Yaskawa INFORM job: X2_104(180,0).JBI

/JOB
//NAME X2_104(180,0)
//POS
///NPOS 389,389,389,11,0,0
///TOOL 0
///POSTYPE PULSE
///PULSE
C00000=-2887,-122912,-116763,204,79921,-300
C00001=105948,-60265,-68612,15471,82266,-26774
C00002=105944,-60303,-65683,15533,80508,-26998
C00003=105943,-60263,-64482,15562,79814,-27086
C00004=105942,-60151,-62762,15605,78849,-27210
C00005=105943,-60263,-64482,15562,79814,-27086
C00006=105943,-60248,-64197,15569,79653,-27107
C00007=105943,-60248,-64195,15569,79652,-27108
C00008=105943,-60248,-64197,15569,79653,-27107
C00009=105943,-60248,-64197,15569,79653,-27107
C00010=105942,-60174,-63048,15598,79008,-27190
C00011=105941,-60184,-63045,15598,79001,-27191
C00012=105942,-60174,-63048,15598,79008,-27190
C00013=105943,-60249,-64198,15569,79653,-27107
C00014=105943,-60263,-64482,15562,79814,-27086
C00015=105944,-60303,-65683,15533,80508,-26998
C00016=105948,-60265,-68612,15471,82266,-26774
C00017=109877,-64973,-75760,9490,93075,-21209
C00018=144619,-68543,-73003,-20989,87470,27722
C00019=149622,-57030,-60721,-30956,83108,29784
C00020=149622,-56790,-58217,-31031,81883,30116
C00021=149622,-56662,-57196,-31066,81398,30250
C00022=149623,-56407,-55393,-31134,80554,30482
C00023=149622,-56662,-57196,-31066,81398,30250
C00024=150587,-55933,-56592,-31222,81757,30533
C00025=149619,-56625,-56981,-31073,81300,30276
C00026=149621,-56633,-56977,-31074,81295,30278
C00027=149622,-56635,-56981,-31074,81296,30278
C00028=149617,-56657,-57316,-31061,81462,30231
C00029=149617,-56657,-57313,-31061,81461,30231
C00030=149617,-56657,-57316,-31061,81462,30231
C00031=149622,-56635,-56981,-31074,81296,30278
C00032=149622,-56662,-57196,-31066,81398,30250
C00033=149622,-56790,-58217,-31031,81883,30116
C00034=149622,-57030,-60721,-30956,83108,29784
C00035=144619,-68543,-73003,-20989,87470,27722
C00036=114895,-83747,-80366,6772,73338,-8124
C00037=115460,-69444,-73725,6516,76534,-7754
C00038=115459,-69304,-70716,6562,74765,-7849
C00039=115458,-69195,-69485,6584,74068,-7887
C00040=115458,-68988,-67720,6614,73094,-7940
C00041=115458,-69195,-69485,6584,74068,-7887
C00042=115458,-69074,-68335,6603,73428,-7921
C00043=115457,-69075,-68332,6603,73425,-7921
C00044=115458,-69074,-68335,6603,73428,-7921
C00045=115458,-69210,-69581,6582,74119,-7884
C00046=115459,-69422,-72626,6532,75874,-7789
C00047=114895,-83747,-80366,6772,73338,-8124
C00048=122568,-82719,-80422,-802,72905,572
C00049=122404,-70386,-74693,-742,75716,497
C00050=122404,-70253,-71692,-748,73937,507
C00051=122404,-70146,-70463,-750,73236,512
C00052=122404,-69945,-68703,-754,72256,518
C00053=122404,-70146,-70463,-750,73236,512
C00054=122403,-69999,-69129,-754,72490,516
C00055=122403,-69999,-69126,-754,72489,516
C00056=122403,-69999,-69129,-754,72490,516
C00057=122426,-71764,-70432,-761,72385,525
C00058=125366,-69810,-69017,-1661,72563,1552
C00059=139732,-60008,-63655,-19169,79951,16701
C00060=138795,-60432,-63881,-18965,79660,16411
C00061=141372,-63440,-66071,-19537,80074,17269
C00062=131414,-76802,-75559,-9437,74661,8207
C00063=122633,-87524,-80325,-832,70378,611
C00064=122404,-70253,-71692,-748,73937,507
C00065=122404,-70386,-74693,-742,75716,497
C00066=122568,-82719,-80422,-802,72905,572
C00067=120793,-80683,-79694,968,73556,-1433
C00068=120782,-70088,-74721,961,75940,-1419
C00069=120781,-69974,-71726,968,74156,-1433
C00070=120781,-69875,-70501,972,73453,-1438
C00071=120781,-69685,-68746,976,72471,-1446
C00072=120781,-69875,-70501,972,73453,-1438
C00073=120781,-69719,-69028,976,72627,-1445
C00074=120781,-69719,-69024,976,72624,-1446
C00075=120781,-69719,-69028,976,72627,-1445
C00076=120781,-69868,-70316,972,73342,-1439
C00077=121987,-69893,-70664,604,73531,-1018
C00078=120781,-69902,-70677,972,73547,-1437
C00079=120781,-69912,-70673,972,73540,-1437
C00080=120781,-69738,-69020,976,72612,-1445
C00081=120781,-69875,-70501,972,73453,-1438
C00082=120781,-69974,-71726,968,74156,-1433
C00083=120782,-70088,-74721,961,75940,-1419
C00084=109767,-94679,-77625,-554,64647,-3819
C00085=110036,-87261,-71666,-642,64793,-3719
C00086=110147,-84282,-69219,-679,64819,-3677
C00087=106931,-83315,-68824,372,65076,-4870
C00088=120553,-76872,-65939,-13890,70696,12122
C00089=123092,-73013,-64238,-16293,73991,15774
C00090=123502,-72820,-64152,-16860,74575,16660
C00091=130441,-60579,-57109,-23338,83277,32357
C00092=128852,-72596,-62262,-22941,75556,33354
C00093=130317,-73839,-64199,-23146,76478,33722
C00094=133782,-77123,-68532,-23639,78364,34645
C00095=137012,-102538,-78858,-24747,73168,36952
C00096=156868,-82779,-69870,-33497,82961,10620
C00097=152555,-67883,-62928,-32980,84120,8538
C00098=153259,-66149,-60215,-33082,83738,8932
C00099=149912,-60899,-55666,-32717,82430,7997
C00100=128127,-81205,-68774,-8858,64404,-8706
C00101=128406,-81696,-69061,-3569,63264,-13044
C00102=126372,-87795,-73203,-2830,62599,-13791
C00103=116888,-93582,-79828,8557,66782,-12634
C00104=92924,-89512,-73118,32406,78401,-8719
C00105=72721,-73373,-69592,26022,86972,-15267
C00106=80895,-52896,-59408,25141,88320,-11942
C00107=83138,-49043,-54251,24862,86564,-11488
C00108=85205,-49270,-53237,24600,85277,-10995
C00109=85821,-49873,-53436,24520,84922,-10841
C00110=95949,-62919,-60694,23037,79963,-8102
C00111=102091,-71911,-65157,19247,73237,-2273
C00112=116516,-77081,-67507,13716,67864,4585
C00113=112851,-78661,-66635,20192,66100,7115
C00114=125798,-85436,-69237,6250,57352,21558
C00115=146063,-75361,-64399,-19160,63709,45094
C00116=156433,-45058,-47672,-31921,84708,61878
C00117=158375,-58932,-51564,-37026,71970,66054
C00118=159846,-59274,-53202,-37172,73275,66233
C00119=163234,-59592,-56142,-37574,76069,66714
C00120=168472,-71553,-64044,-35465,82568,67157
C00121=118088,-113838,-85475,7366,65299,-32947
C00122=118732,-79947,-72555,6808,74639,-32160
C00123=121034,-75641,-67247,6295,73405,-31417
C00124=122088,-73495,-65040,6051,73071,-31063
C00125=121942,-71052,-63825,6072,73586,-31087
C00126=123099,-75779,-64750,4483,66211,-39428
C00127=121321,-81189,-67590,5597,62405,-44748
C00128=118846,-85423,-72852,6459,63648,-45617
C00129=118212,-118410,-84702,7387,54112,-46472
C00130=-871,-167382,-128748,-2443,88873,-10065
C00131=-871,-167382,-128748,-2443,88873,-10065
C00132=57381,82979,10637,-12644,90379,68932
C00133=127807,-61304,-68748,-13816,80064,24242
C00134=125765,-61582,-65964,-13370,77922,23771
C00135=124946,-61609,-64807,-13191,77080,23576
C00136=124950,-61468,-63072,-13241,76110,23683
C00137=124946,-61609,-64807,-13191,77080,23576
C00138=124976,-61587,-64521,-13207,76925,23603
C00139=124980,-61587,-64530,-13208,76931,23604
C00140=124976,-61587,-64521,-13207,76925,23603
C00141=124935,-61591,-64522,-13196,76916,23590
C00142=124937,-61496,-63363,-13229,76268,23661
C00143=123116,-61640,-63435,-12754,75950,23053
C00144=124937,-61496,-63363,-13229,76268,23661
C00145=124935,-61591,-64522,-13196,76916,23590
C00146=124946,-61609,-64807,-13191,77080,23576
C00147=125765,-61582,-65964,-13370,77922,23771
C00148=127807,-61304,-68748,-13816,80064,24242
C00149=123100,-60794,-73195,-8642,92314,18302
C00150=97511,-77513,-76888,20898,84915,-28039
C00151=93556,-58201,-60930,30710,81826,-29583
C00152=93550,-57951,-58428,30804,80607,-29915
C00153=93548,-57820,-57410,30845,80124,-30048
C00154=93546,-57539,-55590,30923,79282,-30278
C00155=93548,-57820,-57410,30845,80124,-30048
C00156=93547,-57790,-57188,30855,80020,-30076
C00157=93545,-57800,-57196,30855,80021,-30077
C00158=93547,-57790,-57188,30855,80020,-30076
C00159=93548,-57786,-57169,30855,80012,-30078
C00160=93543,-57856,-57518,30843,80168,-30037
C00161=93543,-57857,-57528,30842,80172,-30036
C00162=93543,-57856,-57518,30843,80168,-30037
C00163=93548,-57786,-57169,30855,80012,-30078
C00164=93548,-57820,-57410,30845,80124,-30048
C00165=93550,-57951,-58428,30804,80607,-29915
C00166=93556,-58201,-60930,30710,81826,-29583
C00167=97511,-77513,-76888,20898,84915,-28039
C00168=129623,-93566,-83802,-7941,70327,9276
C00169=128126,-69066,-72890,-7284,76011,8392
C00170=128127,-68885,-69881,-7338,74266,8496
C00171=128227,-70585,-69547,-7404,73204,8596
C00172=128227,-70369,-67888,-7439,72303,8652
C00173=128262,-71214,-69852,-7419,73073,8616
C00174=128200,-69934,-68140,-7416,72675,8619
C00175=128127,-68612,-67496,-7384,72949,8576
C00176=128127,-68613,-67489,-7384,72944,8577
C00177=128127,-68764,-68733,-7360,73627,8535
C00178=128126,-69014,-71778,-7303,75358,8431
C00179=129623,-93566,-83802,-7941,70327,9276
C00180=121374,-102449,-87359,-63,66651,180
C00181=121222,-71970,-74483,-14,74388,124
C00182=121222,-71735,-71450,-14,72642,124
C00183=121228,-73354,-70977,-16,71518,126
C00184=121228,-73077,-69260,-16,70604,126
C00185=121230,-73832,-71281,-16,71462,127
C00186=121229,-73317,-69774,-16,70798,128
C00187=121222,-71403,-68866,-14,71222,125
C00188=121222,-71402,-68857,-14,71217,125
C00189=121222,-71370,-68825,-14,71214,125
C00190=121222,-71504,-69842,-14,71771,124
C00191=121222,-71516,-69850,-14,71770,124
C00192=121222,-71504,-69842,-14,71771,124
C00193=121222,-71598,-70490,-14,72121,125
C00194=121222,-71590,-70211,-14,71954,124
C00195=121222,-71735,-71450,-14,72642,124
C00196=121222,-71970,-74483,-14,74388,124
C00197=121374,-102449,-87359,-63,66651,180
C00198=123521,-105913,-88673,-2044,65797,2436
C00199=122862,-71970,-74551,-1739,74528,2064
C00200=122862,-71740,-71520,-1753,72781,2089
C00201=122863,-71596,-70280,-1759,72093,2099
C00202=122863,-71343,-68495,-1768,71124,2113
C00203=122863,-71596,-70280,-1759,72093,2099
C00204=122863,-71387,-68782,-1767,71278,2111
C00205=122863,-71388,-68789,-1767,71282,2111
C00206=122863,-71387,-68782,-1767,71278,2111
C00207=122862,-71560,-70082,-1760,71989,2100
C00208=122862,-71596,-70456,-1758,72201,2098
C00209=122862,-71608,-70465,-1758,72201,2098
C00210=122862,-71596,-70456,-1758,72201,2098
C00211=122862,-71364,-68762,-1767,71278,2111
C00212=122863,-71596,-70280,-1759,72093,2099
C00213=122862,-71740,-71520,-1753,72781,2089
C00214=122862,-71970,-74551,-1739,74528,2064
C00215=133853,-94891,-77624,-322,64195,4510
C00216=133469,-87446,-71679,-193,64361,4366
C00217=133332,-84612,-69279,-149,64338,4316
C00218=136520,-83360,-68727,-1205,64680,5498
C00219=122681,-77523,-66172,13350,69902,-11676
C00220=120168,-73612,-64489,15807,73184,-15339
C00221=112575,-61593,-57739,23052,82443,-32062
C00222=113938,-70945,-61811,22691,76593,-32754
C00223=112608,-75313,-64851,22854,75462,-33489
C00224=109132,-78771,-69243,23377,77292,-34432
C00225=105658,-108562,-80888,24788,70838,-37103
C00226=81640,-97499,-76087,33945,80765,-12609
C00227=90241,-69606,-64048,32870,83199,-8395
C00228=92951,-64963,-58962,32610,81520,-7798
C00229=93939,-63321,-57029,32518,80848,-7597
C00230=125857,-77866,-68310,-6550,68061,3456
C00231=123054,-78148,-68482,-5670,67810,2448
C00232=143027,-65706,-58192,-31754,78539,6334
C00233=144021,-67708,-60230,-31872,79107,6572
C00234=146628,-72736,-65452,-32167,80634,7181
C00235=152532,-96040,-75422,-33296,77968,10353
C00236=170079,-74119,-69784,-26506,86877,15660
C00237=161776,-50684,-58065,-25622,88646,12176
C00238=159526,-46913,-52939,-25338,86859,11731
C00239=158170,-45955,-51438,-25163,86055,11404
C00240=157195,-47475,-52284,-25036,85525,11154
C00241=146543,-61011,-59669,-23472,80213,8306
C00242=141963,-69014,-63758,-20053,74078,2973
C00243=126831,-75909,-66940,-14438,68034,-4018
C00244=130165,-77618,-66175,-20834,66320,-6667
C00245=117599,-84808,-69026,-7184,57298,-20899
C00246=97281,-75815,-64687,18602,62898,-44607
C00247=86271,-46211,-48696,31805,84024,-61698
C00248=85005,-58470,-51696,36499,71620,-65497
C00249=82871,-59517,-53345,37068,72494,-66094
C00250=79472,-59950,-56347,37489,75274,-66588
C00251=72756,-72734,-64617,35623,82237,-67485
C00252=121023,-109349,-83964,-6868,66067,31929
C00253=120934,-78788,-71982,-6517,74337,31434
C00254=118696,-74387,-66630,-5999,73137,30708
C00255=117510,-72864,-64443,-5724,72490,30318
C00256=117903,-69871,-63138,-5800,73250,30422
C00257=117006,-77674,-64461,-4475,61816,43275
C00258=118051,-79909,-67055,-4889,62200,43848
C00259=120454,-84253,-72369,-5752,63392,44701
C00260=120394,-115928,-83972,-6293,54299,45179
C00261=-2019,-116841,-84248,8,53945,-8
C00262=-2019,-116841,-84248,8,53945,-8
C00263=73594,47215,-15331,-17682,89066,63909
C00264=142113,-97158,-104646,-26332,80699,28696
C00265=126900,-111905,-82922,-22333,65135,26241
C00266=123037,-105645,-78013,-21421,64295,24879
C00267=121585,-103154,-76020,-21064,63971,24366
C00268=121574,-101968,-73872,-21184,63301,24491
C00269=121585,-103154,-76020,-21064,63971,24366
C00270=121605,-102291,-74338,-21170,63423,24480
C00271=121584,-98936,-73211,-20991,64381,24287
C00272=121605,-102291,-74338,-21170,63423,24480
C00273=121452,-100284,-74443,-20948,64409,24229
C00274=118901,-100253,-74439,-20311,63782,23339
C00275=121452,-100284,-74443,-20948,64409,24229
C00276=122866,-102731,-76445,-21292,64747,24723
C00277=126621,-108872,-81370,-22171,65621,26033
C00278=121330,-115088,-85498,-358,58030,151
C00279=121291,-106557,-79734,-341,58867,134
C00280=121277,-103287,-77415,-334,59121,127
C00281=121267,-102136,-75285,-334,58400,125
C00282=121277,-103287,-77415,-334,59121,127
C00283=121242,-102632,-75811,-324,58469,116
C00284=121234,-99223,-74662,-318,59514,110
C00285=121242,-102632,-75811,-324,58469,116
C00286=121256,-105876,-78126,-330,58227,122
C00287=121292,-114324,-83876,-346,57425,139
C00288=121322,-115349,-85447,-355,57865,149
C00289=121283,-106809,-79688,-338,58709,131
C00290=121269,-103536,-77371,-332,58965,124
C00291=121259,-102375,-75237,-331,58248,123
C00292=121269,-103536,-77371,-332,58965,124
C00293=121253,-102639,-75604,-329,58338,121
C00294=121245,-99239,-74459,-322,59381,114
C00295=121253,-102639,-75604,-329,58338,121
C00296=121268,-105882,-77919,-334,58096,127
C00297=121305,-114323,-83666,-351,57296,144
C00298=121318,-115477,-85353,-354,57741,148
C00299=121280,-106935,-79598,-338,58589,130
C00300=121266,-103662,-77282,-331,58845,124
C00301=121256,-102495,-75146,-331,58130,122
C00302=121266,-103662,-77282,-331,58845,124
C00303=121259,-102859,-75577,-331,58209,124
C00304=121251,-99462,-74437,-325,59253,117
C00305=121259,-102859,-75577,-331,58209,124
C00306=121274,-106105,-77890,-337,57965,130
C00307=121311,-114553,-83633,-354,57157,147
C00308=121337,-115746,-85310,-361,57577,156
C00309=121297,-107196,-79560,-344,58432,137
C00310=121283,-103917,-77246,-338,58692,131
C00311=121272,-102742,-75106,-337,57980,130
C00312=121283,-103917,-77246,-338,58692,131
C00313=121246,-102874,-75436,-326,58114,118
C00314=121237,-99483,-74299,-320,59157,112
C00315=121246,-102874,-75436,-326,58114,118
C00316=121259,-106119,-77748,-333,57870,124
C00317=121296,-114563,-83488,-348,57063,142
C00318=115780,-112688,-82708,21819,64400,-26075
C00319=119618,-106339,-77769,20890,63616,-24706
C00320=121058,-103816,-75763,20529,63312,-24192
C00321=121048,-102603,-73605,20653,62653,-24321
C00322=121058,-103816,-75763,20529,63312,-24192
C00323=121040,-102752,-73855,20641,62728,-24310
C00324=121038,-99421,-72747,20466,63695,-24129
C00325=121040,-102752,-73855,20641,62728,-24310
C00326=118303,-96965,-72660,22305,67146,-26975
C00327=118267,-92509,-70963,23513,70285,-29122
C00328=120824,-100634,-73993,20495,63883,-24177
C00329=119419,-103098,-76004,20840,64209,-24672
C00330=115684,-109288,-80956,21727,65048,-25985
C00331=96888,-111476,-87068,9061,72855,-9977
C00332=98574,-104492,-81262,8787,72684,-9391
C00333=93909,-110684,-79514,13666,64171,-14539
C00334=141627,-111255,-79468,4808,59529,5267
C00335=116884,-104836,-72389,32528,66157,393
C00336=116227,-100796,-73717,31025,72452,2000
C00337=113714,-107379,-79275,31259,73409,1253
C00338=145516,-110399,-87018,-9521,73555,10095
C00339=143792,-103507,-81225,-9247,73331,9501
C00340=147991,-116725,-79770,-15189,57547,12945
C00341=92805,-108670,-79244,2926,60987,-8726
C00342=125500,-104465,-72202,-33294,65779,-22
C00343=126155,-100219,-73727,-31459,72916,-1934
C00344=128707,-106743,-79266,-31688,73916,-1183
C00345=149163,-107491,-85659,-10054,74646,11300
C00346=147320,-100877,-79905,-9779,74280,10678
C00347=149405,-108030,-78804,-12916,65248,12387
C00348=93726,-109350,-79423,2686,60646,-8385
C00349=95575,-101419,-80230,-67,70891,-7504
C00350=94880,-108692,-86195,76,70825,-7751
C00351=93512,-107502,-86110,9531,74678,-11036
C00352=95285,-100847,-80339,9259,74342,-10434
C00353=91829,-111238,-79018,14022,61540,-13112
C00354=149361,-109410,-78888,-3377,59825,8868
C00355=152861,-110027,-78581,-5464,58492,10359
C00356=146783,-100727,-80168,-430,71345,7655
C00357=147530,-107934,-86130,-582,71316,7920
C00358=147530,-109971,-90893,-577,73200,7911
C00359=147530,-109971,-90893,-577,73200,7911
C00360=129338,-115306,-83649,32043,62659,-1447
C00361=109985,-114895,-67593,57991,58611,-29778
C00362=123189,-110825,-64198,56881,47665,-25598
C00363=123974,-108354,-57257,59191,45569,-26987
C00364=133588,-111477,-65669,41012,44431,-18914
C00365=131723,-121473,-78996,33426,49678,-16861
C00366=131723,-127083,-87093,32500,51454,-16199
C00367=112124,-99575,-74661,44559,72636,-57535
C00368=144481,-87729,-76760,13160,69523,-45180
C00369=143253,-81512,-73231,13426,70725,-45494
C00370=141746,-72876,-67816,13764,72050,-45890
C00371=140405,-91076,-80988,14230,71070,-46496
C00372=147724,-115880,-117962,-4434,76384,7704
C00373=102175,-95850,-84882,-8811,63963,-9409
C00374=106773,-75463,-61467,-29853,53349,18924
C00375=99131,-70118,-56440,-22082,48330,13186
C00376=98320,-68106,-55033,-21545,48270,12812
C00377=98199,-68741,-54193,-21751,47452,12950
C00378=97569,-68978,-50300,-22280,44856,13272
C00379=93899,-57457,-51708,-11926,60791,9289
C00380=97609,-69104,-63179,-12714,63588,10475
C00381=100380,-33173,-52064,-13535,85135,38620
C00382=91620,-26640,-46583,-3556,85730,36721
C00383=94429,-23251,-43461,-7027,86025,37207
C00384=96713,-17180,-36687,-8408,83804,38028
C00385=103963,-23375,-42130,-14397,84680,39883
C00386=111815,-38667,-59152,-16138,88632,42049
C00387=147724,-115880,-117962,-4434,76384,7704
C00388=-2019,-116841,-84248,8,53945,-8
BC00000=780,523905,878730
BC00001=24680,466753,17
BC00002=21091,462611,17
BC00003=19655,460955,17
BC00004=19671,460959,17
BC00005=19655,460955,17
BC00006=19705,460415,17
BC00007=19697,457343,17
BC00008=19705,460415,17
BC00009=19637,460956,17
BC00010=19648,460935,17
BC00011=16462,460942,17
BC00012=19648,460935,17
BC00013=19637,460956,17
BC00014=19655,460955,17
BC00015=21091,462611,17
BC00016=24680,466753,17
BC00017=23714,465651,17
BC00018=75244,465786,17
BC00019=74371,466642,17
BC00020=78995,462188,17
BC00021=80845,460407,17
BC00022=80861,460411,17
BC00023=80845,460407,17
BC00024=81362,460408,17
BC00025=84547,460400,17
BC00026=81362,460408,17
BC00027=80862,466105,17
BC00028=88196,466087,17
BC00029=88188,463015,17
BC00030=88196,466087,17
BC00031=80862,466105,17
BC00032=80845,460407,17
BC00033=78995,462188,17
BC00034=74371,466642,17
BC00035=75244,465786,17
BC00036=130207,468776,17
BC00037=130207,468776,17
BC00038=128970,463491,17
BC00039=128475,461377,17
BC00040=128491,461381,17
BC00041=128475,461377,17
BC00042=126183,462269,17
BC00043=125467,459275,17
BC00044=126183,462269,17
BC00045=126677,464383,17
BC00046=127915,469668,17
BC00047=130207,468776,17
BC00048=334579,467175,17
BC00049=334579,467175,17
BC00050=334594,461751,17
BC00051=334599,459581,17
BC00052=334616,459585,17
BC00053=334599,459581,17
BC00054=334621,459509,17
BC00055=334613,456436,17
BC00056=334621,459509,17
BC00057=326309,462655,17
BC00058=326309,462655,17
BC00059=323407,460034,17
BC00060=323407,460034,17
BC00061=323407,460034,17
BC00062=325115,461032,17
BC00063=334599,459581,17
BC00064=334594,461751,17
BC00065=334579,467175,17
BC00066=334579,467175,17
BC00067=391469,467628,17
BC00068=391469,467628,17
BC00069=391192,462215,17
BC00070=391081,460050,17
BC00071=391097,460054,17
BC00072=391081,460050,17
BC00073=391084,460088,17
BC00074=390911,457021,17
BC00075=391084,460088,17
BC00076=387971,461309,17
BC00077=384628,457146,17
BC00078=387809,456979,17
BC00079=384628,457146,17
BC00080=384826,460381,17
BC00081=391081,460050,17
BC00082=391192,462215,17
BC00083=391469,467628,17
BC00084=363156,441715,38776
BC00085=363156,441715,38776
BC00086=363156,441715,38776
BC00087=363156,441715,38776
BC00088=363156,441715,38776
BC00089=363156,441715,38776
BC00090=363156,441715,38776
BC00091=363156,441715,38776
BC00092=363156,441715,38776
BC00093=363156,441715,38776
BC00094=363156,441715,38776
BC00095=363156,441715,38776
BC00096=338596,448628,25253
BC00097=338596,448628,25253
BC00098=338596,448628,25253
BC00099=338597,448627,25252
BC00100=338597,448627,25252
BC00101=338597,448627,25252
BC00102=338597,448627,25252
BC00103=338597,448627,25252
BC00104=338596,448628,25253
BC00105=96993,454866,20869
BC00106=98278,457002,17644
BC00107=98278,457002,17644
BC00108=98278,457002,17644
BC00109=98278,457002,17644
BC00110=98278,457002,17644
BC00111=98278,457002,17644
BC00112=98278,457002,17644
BC00113=98278,457002,17644
BC00114=98278,457002,17644
BC00115=98278,457002,17644
BC00116=98278,457002,17644
BC00117=98278,457002,17644
BC00118=98278,457002,17644
BC00119=98278,457002,17644
BC00120=96993,454866,20869
BC00121=35692,446449,44492
BC00122=35692,446449,44492
BC00123=35692,446449,44492
BC00124=35692,446449,44492
BC00125=35692,446449,44492
BC00126=35692,446449,44492
BC00127=35692,446449,44492
BC00128=35692,446449,44492
BC00129=35692,446449,44492
BC00130=226112,522070,21179
BC00131=226112,522070,21179
BC00132=201604,630124,773856
BC00133=397680,544373,17
BC00134=397680,461002,17
BC00135=397680,459324,17
BC00136=397680,459307,17
BC00137=397680,459324,17
BC00138=397680,458781,17
BC00139=397680,455709,17
BC00140=397680,458781,17
BC00141=397680,459321,17
BC00142=397680,459287,17
BC00143=397680,459279,17
BC00144=397680,459287,17
BC00145=397680,459321,17
BC00146=397680,459324,17
BC00147=397680,461002,17
BC00148=397680,465197,17
BC00149=397680,464098,17
BC00150=364002,464474,17
BC00151=364885,465316,17
BC00152=360253,460854,17
BC00153=358400,459070,17
BC00154=358395,459053,17
BC00155=358400,459070,17
BC00156=357885,459071,17
BC00157=354700,459079,17
BC00158=357885,459071,17
BC00159=358414,464766,17
BC00160=351078,464787,17
BC00161=351070,461715,17
BC00162=351078,464787,17
BC00163=358414,464766,17
BC00164=358400,459070,17
BC00165=360253,460854,17
BC00166=364885,465316,17
BC00167=364002,464474,17
BC00168=309055,467727,17
BC00169=309055,467727,17
BC00170=310284,462400,17
BC00171=310775,460269,17
BC00172=310770,460253,17
BC00173=310775,460269,17
BC00174=313079,461137,17
BC00175=313780,458140,17
BC00176=313079,461137,17
BC00177=312588,463268,17
BC00178=311359,468595,17
BC00179=309055,467727,17
BC00180=104675,467109,17
BC00181=104675,467109,17
BC00182=104651,461649,17
BC00183=104636,459449,17
BC00184=104636,459449,17
BC00185=104642,459465,17
BC00186=104628,459377,17
BC00187=104620,456305,17
BC00188=104628,459377,17
BC00189=112956,462483,17
BC00190=116212,459519,17
BC00191=113027,459526,17
BC00192=116212,459519,17
BC00193=112864,461621,17
BC00194=104642,459465,17
BC00195=104651,461649,17
BC00196=104675,467109,17
BC00197=104675,467109,17
BC00198=47788,467835,17
BC00199=47788,467835,17
BC00200=48056,462385,17
BC00201=48163,460205,17
BC00202=48157,460188,17
BC00203=48163,460205,17
BC00204=48169,460226,17
BC00205=48326,457158,17
BC00206=48169,460226,17
BC00207=51281,461447,17
BC00208=54599,457272,17
BC00209=51418,457121,17
BC00210=54599,457272,17
BC00211=54429,460489,17
BC00212=48163,460205,17
BC00213=48056,462385,17
BC00214=47788,467835,17
BC00215=75364,442731,32628
BC00216=75364,442731,32628
BC00217=75364,442731,32628
BC00218=75364,442731,32628
BC00219=75364,442731,32628
BC00220=75364,442731,32628
BC00221=75364,442731,32628
BC00222=75364,442731,32628
BC00223=75364,442731,32628
BC00224=75364,442731,32628
BC00225=75364,442731,32628
BC00226=99841,449109,19074
BC00227=99841,449109,19074
BC00228=99841,449109,19074
BC00229=99841,449109,19074
BC00230=99841,449109,19074
BC00231=99841,449109,19074
BC00232=99841,449109,19074
BC00233=99841,449109,19074
BC00234=99841,449109,19074
BC00235=99841,449109,19074
BC00236=339958,454510,16791
BC00237=340496,456637,13010
BC00238=340496,456637,13010
BC00239=340496,456637,13010
BC00240=340496,456637,13010
BC00241=340496,456637,13010
BC00242=340496,456637,13010
BC00243=340496,456637,13010
BC00244=340496,456637,13010
BC00245=340496,456637,13010
BC00246=340496,456637,13010
BC00247=340496,456637,13010
BC00248=340496,456637,13010
BC00249=340496,456637,13010
BC00250=340496,456637,13010
BC00251=339958,454510,16791
BC00252=397680,444887,42686
BC00253=397680,444887,42686
BC00254=397680,444887,42686
BC00255=397680,444887,42686
BC00256=397680,444887,42686
BC00257=397680,444887,42686
BC00258=397680,444887,42686
BC00259=397680,444887,42686
BC00260=397680,444887,42686
BC00261=262396,523905,990511
BC00262=262396,523905,990511
BC00263=128960,592658,1075149
BC00264=336620,434807,1075139
BC00265=336620,389215,1075139
BC00266=336620,389215,1075139
BC00267=336620,389215,1075139
BC00268=336620,389215,1075139
BC00269=336620,389215,1075139
BC00270=336620,389215,1075139
BC00271=336620,389215,1075139
BC00272=336620,389215,1075139
BC00273=336620,389215,1075139
BC00274=336620,389215,1075139
BC00275=336620,389215,1075139
BC00276=336620,389215,1075139
BC00277=336620,389215,1075139
BC00278=314467,401738,1075139
BC00279=314467,401738,1075139
BC00280=314467,401738,1075139
BC00281=314467,401738,1075139
BC00282=314467,401738,1075139
BC00283=314467,401738,1075139
BC00284=314467,401738,1075139
BC00285=314467,401738,1075139
BC00286=314467,401738,1075139
BC00287=314467,401738,1075139
BC00288=250431,402103,1075139
BC00289=250431,402103,1075139
BC00290=250431,402103,1075139
BC00291=250431,402103,1075139
BC00292=250431,402103,1075139
BC00293=250431,402103,1075139
BC00294=250431,402103,1075139
BC00295=250431,402103,1075139
BC00296=250431,402103,1075139
BC00297=250431,402103,1075139
BC00298=181730,402292,1075139
BC00299=181730,402292,1075139
BC00300=181730,402292,1075139
BC00301=181730,402292,1075139
BC00302=181730,402292,1075139
BC00303=181730,402292,1075139
BC00304=181730,402292,1075139
BC00305=181730,402292,1075139
BC00306=181730,402292,1075139
BC00307=181730,402292,1075139
BC00308=120634,402626,1075139
BC00309=120634,402626,1075139
BC00310=120634,402626,1075139
BC00311=120634,402626,1075139
BC00312=120634,402626,1075139
BC00313=120634,402626,1075139
BC00314=120634,402626,1075139
BC00315=120634,402626,1075139
BC00316=120634,402626,1075139
BC00317=120634,402626,1075139
BC00318=98246,390680,1075139
BC00319=98246,390680,1075139
BC00320=98246,390680,1075139
BC00321=98246,390680,1075139
BC00322=98246,390680,1075139
BC00323=98246,390680,1075139
BC00324=98246,390680,1075139
BC00325=98246,390680,1075139
BC00326=98246,390680,1075139
BC00327=98246,390680,1075139
BC00328=98246,390680,1075139
BC00329=98246,390680,1075139
BC00330=98246,390680,1075139
BC00331=102602,381344,1075139
BC00332=102602,381344,1075139
BC00333=102602,381344,1075139
BC00334=102602,381344,1075139
BC00335=102602,381344,1075139
BC00336=102602,381344,1075139
BC00337=102602,381344,1075139
BC00338=332399,380541,1075139
BC00339=332399,380541,1075139
BC00340=332399,380541,1075139
BC00341=332399,380541,1075139
BC00342=332399,380541,1075139
BC00343=332399,380541,1075139
BC00344=332399,380541,1075139
BC00345=143465,382402,1075139
BC00346=143465,382402,1075139
BC00347=143465,382402,1075139
BC00348=143465,382402,1075139
BC00349=143465,382402,1075139
BC00350=143465,382402,1075139
BC00351=291477,381910,1075139
BC00352=291477,381910,1075139
BC00353=291477,381910,1075139
BC00354=291477,381910,1075139
BC00355=291477,381910,1075139
BC00356=291477,381910,1075139
BC00357=291477,381910,1075139
BC00358=291477,381910,1075139
BC00359=130464,381910,1075139
BC00360=130464,381910,1075139
BC00361=130464,381910,1075139
BC00362=130464,381910,1075139
BC00363=130464,381910,1075139
BC00364=130464,381910,1075139
BC00365=130464,381910,1075139
BC00366=130464,381910,1075139
BC00367=130464,381910,1075139
BC00368=130464,381910,1075139
BC00369=130464,381910,1075139
BC00370=130464,381910,1075139
BC00371=130464,381910,1075139
BC00372=291477,429847,1075139
BC00373=290233,429476,1075139
BC00374=290233,429476,1075139
BC00375=290233,429476,1075139
BC00376=290233,429476,1075139
BC00377=290233,429476,1075139
BC00378=290233,429476,1075139
BC00379=290233,429476,1075139
BC00380=290233,429476,1075139
BC00381=290234,429477,1075136
BC00382=290234,429477,1075136
BC00383=290234,429477,1075136
BC00384=290234,429477,1075136
BC00385=290234,429477,1075136
BC00386=290234,429477,1075136
BC00387=291477,429847,1075139
BC00388=262396,523905,990511
EC00000=-1596313,-183832
EC00001=-1596313,-183832
EC00002=-1596313,-183832
EC00003=-1596313,-183832
EC00004=-1596313,-183832
EC00005=-1596313,-183832
EC00006=-1596313,-183832
EC00007=-1596313,-183832
EC00008=-1596313,-183832
EC00009=-1596313,-183832
EC00010=-1596313,-183832
EC00011=-1596313,-183832
EC00012=-1596313,-183832
EC00013=-1596313,-183832
EC00014=-1596313,-183832
EC00015=-1596313,-183832
EC00016=-1596313,-183832
EC00017=-1596313,-183832
EC00018=-1596313,-183832
EC00019=-1596313,-183832
EC00020=-1596313,-183832
EC00021=-1596313,-183832
EC00022=-1596313,-183832
EC00023=-1596313,-183832
EC00024=-1596313,-183832
EC00025=-1596313,-183832
EC00026=-1596313,-183832
EC00027=-1596313,-183832
EC00028=-1596313,-183832
EC00029=-1596313,-183832
EC00030=-1596313,-183832
EC00031=-1596313,-183832
EC00032=-1596313,-183832
EC00033=-1596313,-183832
EC00034=-1596313,-183832
EC00035=-1596313,-183832
EC00036=-1596313,-183832
EC00037=-1596313,-183832
EC00038=-1596313,-183832
EC00039=-1596313,-183832
EC00040=-1596313,-183832
EC00041=-1596313,-183832
EC00042=-1596313,-183832
EC00043=-1596313,-183832
EC00044=-1596313,-183832
EC00045=-1596313,-183832
EC00046=-1596313,-183832
EC00047=-1596313,-183832
EC00048=-1596313,-183832
EC00049=-1596313,-183832
EC00050=-1596313,-183832
EC00051=-1596313,-183832
EC00052=-1596313,-183832
EC00053=-1596313,-183832
EC00054=-1596313,-183832
EC00055=-1596313,-183832
EC00056=-1596313,-183832
EC00057=-1596313,-183832
EC00058=-1596313,-183832
EC00059=-1596313,-183832
EC00060=-1596313,-183832
EC00061=-1596313,-183832
EC00062=-1596313,-183832
EC00063=-1596313,-183832
EC00064=-1596313,-183832
EC00065=-1596313,-183832
EC00066=-1596313,-183832
EC00067=-1596313,-183832
EC00068=-1596313,-183832
EC00069=-1596313,-183832
EC00070=-1596313,-183832
EC00071=-1596313,-183832
EC00072=-1596313,-183832
EC00073=-1596313,-183832
EC00074=-1596313,-183832
EC00075=-1596313,-183832
EC00076=-1596313,-183832
EC00077=-1596313,-183832
EC00078=-1596313,-183832
EC00079=-1596313,-183832
EC00080=-1596313,-183832
EC00081=-1596313,-183832
EC00082=-1596313,-183832
EC00083=-1596313,-183832
EC00084=-1596313,-183832
EC00085=-1596313,-183832
EC00086=-1596313,-183832
EC00087=-1596313,-183832
EC00088=-1596313,-183832
EC00089=-1596313,-183832
EC00090=-1596313,-183832
EC00091=-1596313,-183832
EC00092=-1596313,-183832
EC00093=-1596313,-183832
EC00094=-1596313,-183832
EC00095=-1596313,-183832
EC00096=-1596313,-183832
EC00097=-1596313,-183832
EC00098=-1596313,-183832
EC00099=-1596312,-183832
EC00100=-1596312,-183832
EC00101=-1596312,-183832
EC00102=-1596312,-183832
EC00103=-1596312,-183832
EC00104=-1596313,-183832
EC00105=-1596313,-183832
EC00106=-1596313,-183832
EC00107=-1596313,-183832
EC00108=-1596313,-183832
EC00109=-1596313,-183832
EC00110=-1596313,-183832
EC00111=-1596313,-183832
EC00112=-1596313,-183832
EC00113=-1596313,-183832
EC00114=-1596313,-183832
EC00115=-1596313,-183832
EC00116=-1596313,-183832
EC00117=-1596313,-183832
EC00118=-1596313,-183832
EC00119=-1596313,-183832
EC00120=-1596313,-183832
EC00121=-1596313,-183832
EC00122=-1596313,-183832
EC00123=-1596313,-183832
EC00124=-1596313,-183832
EC00125=-1596313,-183832
EC00126=-1596313,-183832
EC00127=-1596313,-183832
EC00128=-1596313,-183832
EC00129=-1596313,-183832
EC00130=-1596313,-183832
EC00131=-1596313,-1296783
EC00132=-1596313,-1296783
EC00133=-1596313,-1296783
EC00134=-1596313,-1296783
EC00135=-1596313,-1296783
EC00136=-1596313,-1296783
EC00137=-1596313,-1296783
EC00138=-1596313,-1296783
EC00139=-1596313,-1296783
EC00140=-1596313,-1296783
EC00141=-1596313,-1296783
EC00142=-1596313,-1296783
EC00143=-1596313,-1296783
EC00144=-1596313,-1296783
EC00145=-1596313,-1296783
EC00146=-1596313,-1296783
EC00147=-1596313,-1296783
EC00148=-1596313,-1296783
EC00149=-1596313,-1296783
EC00150=-1596313,-1296783
EC00151=-1596313,-1296783
EC00152=-1596313,-1296783
EC00153=-1596313,-1296783
EC00154=-1596313,-1296783
EC00155=-1596313,-1296783
EC00156=-1596313,-1296783
EC00157=-1596313,-1296783
EC00158=-1596313,-1296783
EC00159=-1596313,-1296783
EC00160=-1596313,-1296783
EC00161=-1596313,-1296783
EC00162=-1596313,-1296783
EC00163=-1596313,-1296783
EC00164=-1596313,-1296783
EC00165=-1596313,-1296783
EC00166=-1596313,-1296783
EC00167=-1596313,-1296783
EC00168=-1596313,-1296783
EC00169=-1596313,-1296783
EC00170=-1596313,-1296783
EC00171=-1596313,-1296783
EC00172=-1596313,-1296783
EC00173=-1596313,-1296783
EC00174=-1596313,-1296783
EC00175=-1596313,-1296783
EC00176=-1596313,-1296783
EC00177=-1596313,-1296783
EC00178=-1596313,-1296783
EC00179=-1596313,-1296783
EC00180=-1596313,-1296783
EC00181=-1596313,-1296783
EC00182=-1596313,-1296783
EC00183=-1596313,-1296783
EC00184=-1596313,-1296783
EC00185=-1596313,-1296783
EC00186=-1596313,-1296783
EC00187=-1596313,-1296783
EC00188=-1596313,-1296783
EC00189=-1596313,-1296783
EC00190=-1596313,-1296783
EC00191=-1596313,-1296783
EC00192=-1596313,-1296783
EC00193=-1596313,-1296783
EC00194=-1596313,-1296783
EC00195=-1596313,-1296783
EC00196=-1596313,-1296783
EC00197=-1596313,-1296783
EC00198=-1596313,-1296783
EC00199=-1596313,-1296783
EC00200=-1596313,-1296783
EC00201=-1596313,-1296783
EC00202=-1596313,-1296783
EC00203=-1596313,-1296783
EC00204=-1596313,-1296783
EC00205=-1596313,-1296783
EC00206=-1596313,-1296783
EC00207=-1596313,-1296783
EC00208=-1596313,-1296783
EC00209=-1596313,-1296783
EC00210=-1596313,-1296783
EC00211=-1596313,-1296783
EC00212=-1596313,-1296783
EC00213=-1596313,-1296783
EC00214=-1596313,-1296783
EC00215=-1596313,-1296783
EC00216=-1596313,-1296783
EC00217=-1596313,-1296783
EC00218=-1596313,-1296783
EC00219=-1596313,-1296783
EC00220=-1596313,-1296783
EC00221=-1596313,-1296783
EC00222=-1596313,-1296783
EC00223=-1596313,-1296783
EC00224=-1596313,-1296783
EC00225=-1596313,-1296783
EC00226=-1596313,-1296783
EC00227=-1596313,-1296783
EC00228=-1596313,-1296783
EC00229=-1596313,-1296783
EC00230=-1596313,-1296783
EC00231=-1596313,-1296783
EC00232=-1596313,-1296783
EC00233=-1596313,-1296783
EC00234=-1596313,-1296783
EC00235=-1596313,-1296783
EC00236=-1596313,-1296783
EC00237=-1596313,-1296783
EC00238=-1596313,-1296783
EC00239=-1596313,-1296783
EC00240=-1596313,-1296783
EC00241=-1596313,-1296783
EC00242=-1596313,-1296783
EC00243=-1596313,-1296783
EC00244=-1596313,-1296783
EC00245=-1596313,-1296783
EC00246=-1596313,-1296783
EC00247=-1596313,-1296783
EC00248=-1596313,-1296783
EC00249=-1596313,-1296783
EC00250=-1596313,-1296783
EC00251=-1596313,-1296783
EC00252=-1596313,-1296783
EC00253=-1596313,-1296783
EC00254=-1596313,-1296783
EC00255=-1596313,-1296783
EC00256=-1596313,-1296783
EC00257=-1596313,-1296783
EC00258=-1596313,-1296783
EC00259=-1596313,-1296783
EC00260=-1596313,-1296783
EC00261=-1596313,-1296783
EC00262=-1596313,372643
EC00263=-1492805,372643
EC00264=-1330261,372643
EC00265=-1330261,372643
EC00266=-1330261,372643
EC00267=-1330261,372643
EC00268=-1330261,372643
EC00269=-1330261,372643
EC00270=-1330261,372643
EC00271=-1330261,372643
EC00272=-1330261,372643
EC00273=-1330261,372643
EC00274=-1330261,372643
EC00275=-1330261,372643
EC00276=-1330261,372643
EC00277=-1330261,372643
EC00278=-1330261,372643
EC00279=-1330261,372643
EC00280=-1330261,372643
EC00281=-1330261,372643
EC00282=-1330261,372643
EC00283=-1330261,372643
EC00284=-1330261,372643
EC00285=-1330261,372643
EC00286=-1330261,372643
EC00287=-1330261,372643
EC00288=-1330261,372643
EC00289=-1330261,372643
EC00290=-1330261,372643
EC00291=-1330261,372643
EC00292=-1330261,372643
EC00293=-1330261,372643
EC00294=-1330261,372643
EC00295=-1330261,372643
EC00296=-1330261,372643
EC00297=-1330261,372643
EC00298=-1330261,372643
EC00299=-1330261,372643
EC00300=-1330261,372643
EC00301=-1330261,372643
EC00302=-1330261,372643
EC00303=-1330261,372643
EC00304=-1330261,372643
EC00305=-1330261,372643
EC00306=-1330261,372643
EC00307=-1330261,372643
EC00308=-1330261,372643
EC00309=-1330261,372643
EC00310=-1330261,372643
EC00311=-1330261,372643
EC00312=-1330261,372643
EC00313=-1330261,372643
EC00314=-1330261,372643
EC00315=-1330261,372643
EC00316=-1330261,372643
EC00317=-1330261,372643
EC00318=-1330261,372643
EC00319=-1330261,372643
EC00320=-1330261,372643
EC00321=-1330261,372643
EC00322=-1330261,372643
EC00323=-1330261,372643
EC00324=-1330261,372643
EC00325=-1330261,372643
EC00326=-1330261,372643
EC00327=-1330261,372643
EC00328=-1330261,372643
EC00329=-1330261,372643
EC00330=-1330261,372643
EC00331=-1330261,372643
EC00332=-1330261,372643
EC00333=-1330261,372643
EC00334=-1330261,372643
EC00335=-1330261,372643
EC00336=-1330261,372643
EC00337=-1330261,372643
EC00338=-1330261,372643
EC00339=-1330261,372643
EC00340=-1330261,372643
EC00341=-1330261,372643
EC00342=-1330261,372643
EC00343=-1330261,372643
EC00344=-1330261,372643
EC00345=-1330261,372643
EC00346=-1330261,372643
EC00347=-1330261,372643
EC00348=-1330261,372643
EC00349=-1330261,372643
EC00350=-1330261,372643
EC00351=-1330261,372643
EC00352=-1330261,372643
EC00353=-1330261,372643
EC00354=-1330261,372643
EC00355=-1330261,372643
EC00356=-1330261,372643
EC00357=-1330261,372643
EC00358=-1330261,372643
EC00359=-1330261,372643
EC00360=-1330261,372643
EC00361=-1330261,372643
EC00362=-1330261,372643
EC00363=-1330261,372643
EC00364=-1330261,372643
EC00365=-1330261,372643
EC00366=-1330261,372643
EC00367=-1330261,372643
EC00368=-1330261,372643
EC00369=-1330261,372643
EC00370=-1330261,372643
EC00371=-1330261,372643
EC00372=-1330261,372643
EC00373=-1330261,372643
EC00374=-1330261,372643
EC00375=-1330261,372643
EC00376=-1330261,372643
EC00377=-1330261,372643
EC00378=-1330261,372643
EC00379=-1330261,372643
EC00380=-1330261,372643
EC00381=-1330262,372643
EC00382=-1330262,372643
EC00383=-1330262,372643
EC00384=-1330262,372643
EC00385=-1330262,372643
EC00386=-1330262,372643
EC00387=-1330261,372643
EC00388=-1596313,372643
///POSTYPE BASE
///RECTAN
///RCONF 0,0,0,0,1,0,0,0,0,0,0,0,0,0,0,0,0,0,0,0,0,0,0,0
P00006=2.006,1.622,-0.565,0.0000,0.0000,0.0000
P00021=0.073,2.058,-0.109,0.0000,0.0000,0.0000
P00022=2.006,1.622,-0.565,0.0000,0.0000,0.0000
///RCONF 0,0,0,0,0,0,0,0,0,0,0,0,0,0,0,0,0,0,0,0,0,0,0,0
P00023=-2.957,-4.083,2.762,0.0000,0.0000,0.0000
P00024=-1.466,-0.226,-0.419,0.0000,0.0000,0.0000
P00025=3.643,0.007,-2.585,0.0000,0.0000,0.0000
P00031=-0.170,0.039,-0.647,0.0000,0.0000,0.0000
P00032=-0.423,0.157,3.222,0.0000,0.0000,0.0000
P00033=0.854,-1.099,3.047,0.0000,0.0000,0.0000
///RCONF 0,0,0,0,1,0,0,0,0,0,0,0,0,0,0,0,0,0,0,0,0,0,0,0
P00034=-8.151,9.743,-4.393,0.0000,0.0000,0.0000
///RCONF 0,0,0,0,0,0,0,0,0,0,0,0,0,0,0,0,0,0,0,0,0,0,0,0
P00035=0.390,-0.027,1.040,0.0000,0.0000,0.0000
//INST
///DATE 2024/12/19 13:03
///ATTR SC,RW
///GROUP1 RB1,BS1
///GROUP2 ST1
NOP
'X2_104(180,0)
MOVJ C00000 BC00000 VJ=100.00  +MOVJ EC00000 VJ=100.00
'Path S4732
SFTOF3D
MOVJ C00001 BC00001 VJ=100.00  +MOVJ EC00001 VJ=100.00
MOVL C00002 BC00002 V=800.0  +MOVJ EC00002 VJ=100.00
SMOVL C00003 BC00003 V=166.7  +MOVJ EC00003
SREFP 3 C00004 BC00004  +REFP EC00004
CALL JOB:SEARCH-R1-S13D
SET P025 P006
SFTON3D P025
SMOVL C00005 BC00005 V=166.7  +MOVJ EC00005
SMOVL C00006 BC00006 V=166.7  +MOVJ EC00006
SREFP 3 C00007 BC00007  +REFP EC00007
CALL JOB:SEARCH-R1-S13D
SET P025 P006
SFTON3D P025
SMOVL C00008 BC00008 V=166.7  +MOVJ EC00008
SMOVL C00009 BC00009 V=166.7  +MOVJ EC00009
SMOVL C00010 BC00010 V=166.7  +MOVJ EC00010
SREFP 3 C00011 BC00011  +REFP EC00011
CALL JOB:SEARCH-R1-S13D
SET P025 P006
SFTON3D P025
SMOVL C00012 BC00012 V=166.7  +MOVJ EC00012
SMOVL C00013 BC00013 V=166.7  +MOVJ EC00013
SMOVL C00014 BC00014 V=166.7  +MOVJ EC00014
MOVL C00015 BC00015 V=800.0  +MOVJ EC00015 VJ=100.00
MOVL C00016 BC00016 V=1000.0  +MOVJ EC00016 VJ=100.00
'EndPath S4732
MOVJ C00017 BC00017 VJ=100.00  +MOVJ EC00017 VJ=100.00
MOVJ C00018 BC00018 VJ=100.00  +MOVJ EC00018 VJ=100.00
'Path S4733
SFTOF3D
MOVJ C00019 BC00019 VJ=100.00  +MOVJ EC00019 VJ=100.00
MOVL C00020 BC00020 V=800.0  +MOVJ EC00020 VJ=100.00
SMOVL C00021 BC00021 V=166.7  +MOVJ EC00021
SREFP 3 C00022 BC00022  +REFP EC00022
CALL JOB:SEARCH-R1-S13D
SET P024 P006
SFTON3D P024
SMOVL C00023 BC00023 V=166.7  +MOVJ EC00023
SMOVL C00024 BC00024 V=166.7  +MOVJ EC00024
SREFP 3 C00025 BC00025  +REFP EC00025
CALL JOB:SEARCH-R1-S13D
SET P024 P006
SFTON3D P024
SMOVL C00026 BC00026 V=166.7  +MOVJ EC00026
SMOVL C00027 BC00027 V=166.7  +MOVJ EC00027
SMOVL C00028 BC00028 V=166.7  +MOVJ EC00028
SREFP 3 C00029 BC00029  +REFP EC00029
CALL JOB:SEARCH-R1-S13D
SET P024 P006
SFTON3D P024
SMOVL C00030 BC00030 V=166.7  +MOVJ EC00030
SMOVL C00031 BC00031 V=166.7  +MOVJ EC00031
SMOVL C00032 BC00032 V=166.7  +MOVJ EC00032
MOVL C00033 BC00033 V=800.0  +MOVJ EC00033 VJ=100.00
MOVL C00034 BC00034 V=1000.0  +MOVJ EC00034 VJ=100.00
'EndPath S4733
MOVJ C00035 BC00035 VJ=100.00  +MOVJ EC00035 VJ=100.00
MOVJ C00036 BC00036 VJ=100.00  +MOVJ EC00036 VJ=100.00
'Path S4734
SFTOF3D
MOVJ C00037 BC00037 VJ=100.00  +MOVJ EC00037 VJ=100.00
MOVL C00038 BC00038 V=800.0  +MOVJ EC00038 VJ=100.00
SMOVL C00039 BC00039 V=166.7  +MOVJ EC00039
SREFP 3 C00040 BC00040  +REFP EC00040
CALL JOB:SEARCH-R1-S13D
SET P023 P006
SFTON3D P023
SMOVL C00041 BC00041 V=166.7  +MOVJ EC00041
SMOVL C00042 BC00042 V=166.7  +MOVJ EC00042
SREFP 3 C00043 BC00043  +REFP EC00043
CALL JOB:SEARCH-R1-S13D
SET P023 P006
SFTON3D P023
SMOVL C00044 BC00044 V=166.7  +MOVJ EC00044
MOVL C00045 BC00045 V=800.0  +MOVJ EC00045 VJ=100.00
MOVL C00046 BC00046 V=1000.0  +MOVJ EC00046 VJ=100.00
'EndPath S4734
MOVJ C00047 BC00047 VJ=100.00  +MOVJ EC00047 VJ=100.00
MOVJ C00048 BC00048 VJ=100.00  +MOVJ EC00048 VJ=100.00
'Path S4735
SFTOF3D
MOVJ C00049 BC00049 VJ=100.00  +MOVJ EC00049 VJ=100.00
MOVL C00050 BC00050 V=800.0  +MOVJ EC00050 VJ=100.00
SMOVL C00051 BC00051 V=166.7  +MOVJ EC00051
SREFP 3 C00052 BC00052  +REFP EC00052
CALL JOB:SEARCH-R1-S13D
SET P022 P006
SFTON3D P022
SMOVL C00053 BC00053 V=166.7  +MOVJ EC00053
SMOVL C00054 BC00054 V=166.7  +MOVJ EC00054
SREFP 3 C00055 BC00055  +REFP EC00055
CALL JOB:SEARCH-R1-S13D
SET P022 P006
SFTON3D P022
SMOVL C00056 BC00056 V=166.7  +MOVJ EC00056
SMOVL C00057 BC00057 V=166.7  +MOVJ EC00057
SMOVL C00058 BC00058 V=133.3  +MOVJ EC00058
SMOVL C00059 BC00059 V=166.7  +MOVJ EC00059
SREFP 3 C00060 BC00060  +REFP EC00060
CALL JOB:SEARCH-R1-S13D
SET P022 P006
SFTON3D P022
SMOVL C00061 BC00061 V=166.7  +MOVJ EC00061
SMOVL C00062 BC00062 V=166.7  +MOVJ EC00062
SMOVL C00063 BC00063 V=166.7  +MOVJ EC00063
MOVL C00064 BC00064 V=800.0  +MOVJ EC00064 VJ=100.00
MOVL C00065 BC00065 V=1000.0  +MOVJ EC00065 VJ=100.00
'EndPath S4735
MOVJ C00066 BC00066 VJ=100.00  +MOVJ EC00066 VJ=100.00
MOVJ C00067 BC00067 VJ=100.00  +MOVJ EC00067 VJ=100.00
'Path S4736
SFTOF3D
MOVJ C00068 BC00068 VJ=100.00  +MOVJ EC00068 VJ=100.00
MOVL C00069 BC00069 V=800.0  +MOVJ EC00069 VJ=100.00
SMOVL C00070 BC00070 V=166.7  +MOVJ EC00070
SREFP 3 C00071 BC00071  +REFP EC00071
CALL JOB:SEARCH-R1-S13D
SET P021 P006
SFTON3D P021
SMOVL C00072 BC00072 V=166.7  +MOVJ EC00072
SMOVL C00073 BC00073 V=166.7  +MOVJ EC00073
SREFP 3 C00074 BC00074  +REFP EC00074
CALL JOB:SEARCH-R1-S13D
SET P021 P006
SFTON3D P021
SMOVL C00075 BC00075 V=166.7  +MOVJ EC00075
SMOVL C00076 BC00076 V=166.7  +MOVJ EC00076
SMOVL C00077 BC00077 V=166.7  +MOVJ EC00077
SREFP 3 C00078 BC00078  +REFP EC00078
CALL JOB:SEARCH-R1-S13D
SET P021 P006
SFTON3D P021
SMOVL C00079 BC00079 V=166.7  +MOVJ EC00079
SMOVL C00080 BC00080 V=166.7  +MOVJ EC00080
SMOVL C00081 BC00081 V=166.7  +MOVJ EC00081
MOVL C00082 BC00082 V=800.0  +MOVJ EC00082 VJ=100.00
MOVL C00083 BC00083 V=1000.0  +MOVJ EC00083 VJ=100.00
'EndPath S4736
'Path W4732
SFTOF3D
SFTON3D P021
MOVJ C00084 BC00084 VJ=100.00  +MOVJ EC00084 VJ=100.00
SMOVL C00085 BC00085 V=800.0  +MOVJ EC00085
SMOVL C00086 BC00086 V=150.0 PL=0  +MOVJ EC00086
MACRO1 MJ#(0) ARGF14
ARCON
SMOVL C00087 BC00087 V=10.8  +MOVJ EC00087
SMOVL C00088 BC00088 V=11.7  +MOVJ EC00088
SMOVL C00089 BC00089 V=11.7  +MOVJ EC00089
SMOVL C00090 BC00090 V=12.5  +MOVJ EC00090
SMOVL C00091 BC00091 V=12.5  +MOVJ EC00091
SMOVL C00092 BC00092 V=12.5  +MOVJ EC00092
ARCOF
SMOVL C00093 BC00093 V=800.0  +MOVJ EC00093
SMOVL C00094 BC00094 V=1000.0  +MOVJ EC00094
SFTOF3D
'EndPath W4732
MOVJ C00095 BC00095 VJ=100.00  +MOVJ EC00095 VJ=100.00
MOVJ C00096 BC00096 VJ=100.00  +MOVJ EC00096 VJ=100.00
'Path W4737
SFTOF3D
SFTON3D P022
MOVJ C00097 BC00097 VJ=100.00  +MOVJ EC00097 VJ=100.00
SMOVL C00098 BC00098 V=800.0  +MOVJ EC00098
SMOVL C00099 BC00099 V=150.0 PL=0  +MOVJ EC00099
ARCON
SMOVL C00100 BC00100 V=10.0  +MOVJ EC00100
SMOVL C00101 BC00101 V=10.0  +MOVJ EC00101
ARCOF
SMOVL C00102 BC00102 V=800.0  +MOVJ EC00102
SMOVL C00103 BC00103 V=1000.0  +MOVJ EC00103
SFTOF3D
'EndPath W4737
MOVJ C00104 BC00104 VJ=100.00  +MOVJ EC00104 VJ=100.00
MOVJ C00105 BC00105 VJ=100.00  +MOVJ EC00105 VJ=100.00
'Path W4738
SFTOF3D
SFTON3D P023
MOVJ C00106 BC00106 VJ=100.00  +MOVJ EC00106 VJ=100.00
SMOVL C00107 BC00107 V=800.0  +MOVJ EC00107
SMOVL C00108 BC00108 V=150.0 PL=0  +MOVJ EC00108
ARCON
SMOVL C00109 BC00109 V=10.3  +MOVJ EC00109
SMOVL C00110 BC00110 V=10.3  +MOVJ EC00110
SMOVL C00111 BC00111 V=10.8  +MOVJ EC00111
SFTON3D P024
SMOVL C00112 BC00112 V=10.8  +MOVJ EC00112
SMOVL C00113 BC00113 V=10.8  +MOVJ EC00113
SMOVL C00114 BC00114 V=10.8  +MOVJ EC00114
SMOVL C00115 BC00115 V=10.8  +MOVJ EC00115
SMOVL C00116 BC00116 V=10.8  +MOVJ EC00116
SMOVL C00117 BC00117 V=10.0  +MOVJ EC00117
ARCOF
SMOVL C00118 BC00118 V=800.0  +MOVJ EC00118
SMOVL C00119 BC00119 V=1000.0  +MOVJ EC00119
SFTOF3D
'EndPath W4738
MOVJ C00120 BC00120 VJ=100.00  +MOVJ EC00120 VJ=100.00
MOVJ C00121 BC00121 VJ=100.00  +MOVJ EC00121 VJ=100.00
'Path W4739
SFTOF3D
SFTON3D P025
MOVJ C00122 BC00122 VJ=100.00  +MOVJ EC00122 VJ=100.00
SMOVL C00123 BC00123 V=800.0  +MOVJ EC00123
SMOVL C00124 BC00124 V=150.0 PL=0  +MOVJ EC00124
ARCON
SMOVL C00125 BC00125 V=8.3  +MOVJ EC00125
SMOVL C00126 BC00126 V=8.3  +MOVJ EC00126
ARCOF
SMOVL C00127 BC00127 V=800.0  +MOVJ EC00127
SMOVL C00128 BC00128 V=1000.0  +MOVJ EC00128
SFTOF3D
'EndPath W4739
MOVJ C00129 BC00129 VJ=100.00  +MOVJ EC00129 VJ=100.00
'
MOVJ C00130 BC00130 VJ=100.00  +MOVJ EC00130 VJ=100.00
MOVJ C00131 BC00131 VJ=100.00  +MOVJ EC00131 VJ=100.00
'Path S4745
SFTOF3D
CALL JOB:CLEAN-R1_KM_NEW
MOVJ C00132 BC00132 VJ=50.00  +MOVJ EC00132 VJ=50.00
MOVJ C00133 BC00133 VJ=100.00  +MOVJ EC00133 VJ=100.00
SFTOF3D
MOVL C00134 BC00134 V=800.0  +MOVJ EC00134 VJ=100.00
SMOVL C00135 BC00135 V=166.7  +MOVJ EC00135
SREFP 3 C00136 BC00136  +REFP EC00136
CALL JOB:SEARCH-R1-S13D
SET P025 P006
SFTON3D P025
SMOVL C00137 BC00137 V=166.7  +MOVJ EC00137
SMOVL C00138 BC00138 V=166.7  +MOVJ EC00138
SREFP 3 C00139 BC00139  +REFP EC00139
CALL JOB:SEARCH-R1-S13D
SET P025 P006
SFTON3D P025
SMOVL C00140 BC00140 V=166.7  +MOVJ EC00140
SMOVL C00141 BC00141 V=166.7  +MOVJ EC00141
SMOVL C00142 BC00142 V=166.7  +MOVJ EC00142
SREFP 3 C00143 BC00143  +REFP EC00143
CALL JOB:SEARCH-R1-S13D
SET P025 P006
SFTON3D P025
SMOVL C00144 BC00144 V=166.7  +MOVJ EC00144
SMOVL C00145 BC00145 V=166.7  +MOVJ EC00145
SMOVL C00146 BC00146 V=166.7  +MOVJ EC00146
MOVL C00147 BC00147 V=800.0  +MOVJ EC00147 VJ=100.00
MOVL C00148 BC00148 V=1000.0  +MOVJ EC00148 VJ=100.00
'EndPath S4745
MOVJ C00149 BC00149 VJ=100.00  +MOVJ EC00149 VJ=100.00
MOVJ C00150 BC00150 VJ=100.00  +MOVJ EC00150 VJ=100.00
'Path S4744
SFTOF3D
MOVJ C00151 BC00151 VJ=100.00  +MOVJ EC00151 VJ=100.00
MOVL C00152 BC00152 V=800.0  +MOVJ EC00152 VJ=100.00
SMOVL C00153 BC00153 V=166.7  +MOVJ EC00153
SREFP 3 C00154 BC00154  +REFP EC00154
CALL JOB:SEARCH-R1-S13D
SET P024 P006
SFTON3D P024
SMOVL C00155 BC00155 V=166.7  +MOVJ EC00155
SMOVL C00156 BC00156 V=166.7  +MOVJ EC00156
SREFP 3 C00157 BC00157  +REFP EC00157
CALL JOB:SEARCH-R1-S13D
SET P024 P006
SFTON3D P024
SMOVL C00158 BC00158 V=166.7  +MOVJ EC00158
SMOVL C00159 BC00159 V=166.7  +MOVJ EC00159
SMOVL C00160 BC00160 V=166.7  +MOVJ EC00160
SREFP 3 C00161 BC00161  +REFP EC00161
CALL JOB:SEARCH-R1-S13D
SET P024 P006
SFTON3D P024
SMOVL C00162 BC00162 V=166.7  +MOVJ EC00162
SMOVL C00163 BC00163 V=166.7  +MOVJ EC00163
SMOVL C00164 BC00164 V=166.7  +MOVJ EC00164
MOVL C00165 BC00165 V=800.0  +MOVJ EC00165 VJ=100.00
MOVL C00166 BC00166 V=1000.0  +MOVJ EC00166 VJ=100.00
'EndPath S4744
MOVJ C00167 BC00167 VJ=100.00  +MOVJ EC00167 VJ=100.00
MOVJ C00168 BC00168 VJ=100.00  +MOVJ EC00168 VJ=100.00
'Path S4743
SFTOF3D
MOVJ C00169 BC00169 VJ=100.00  +MOVJ EC00169 VJ=100.00
MOVL C00170 BC00170 V=800.0  +MOVJ EC00170 VJ=100.00
SMOVL C00171 BC00171 V=166.7  +MOVJ EC00171
SREFP 3 C00172 BC00172  +REFP EC00172
CALL JOB:SEARCH-R1-S13D
SET P023 P006
SFTON3D P023
SMOVL C00173 BC00173 V=166.7  +MOVJ EC00173
SMOVL C00174 BC00174 V=166.7  +MOVJ EC00174
SREFP 3 C00175 BC00175  +REFP EC00175
CALL JOB:SEARCH-R1-S13D
SET P023 P006
SFTON3D P023
SMOVL C00176 BC00176 V=166.7  +MOVJ EC00176
MOVL C00177 BC00177 V=800.0  +MOVJ EC00177 VJ=100.00
MOVL C00178 BC00178 V=1000.0  +MOVJ EC00178 VJ=100.00
'EndPath S4743
MOVJ C00179 BC00179 VJ=100.00  +MOVJ EC00179 VJ=100.00
MOVJ C00180 BC00180 VJ=100.00  +MOVJ EC00180 VJ=100.00
'Path S4742
SFTOF3D
MOVJ C00181 BC00181 VJ=100.00  +MOVJ EC00181 VJ=100.00
MOVL C00182 BC00182 V=800.0  +MOVJ EC00182 VJ=100.00
SMOVL C00183 BC00183 V=166.7  +MOVJ EC00183
SREFP 3 C00184 BC00184  +REFP EC00184
CALL JOB:SEARCH-R1-S13D
SET P022 P006
SFTON3D P022
SMOVL C00185 BC00185 V=166.7  +MOVJ EC00185
SMOVL C00186 BC00186 V=166.7  +MOVJ EC00186
SREFP 3 C00187 BC00187  +REFP EC00187
CALL JOB:SEARCH-R1-S13D
SET P022 P006
SFTON3D P022
SMOVL C00188 BC00188 V=166.7  +MOVJ EC00188
SMOVL C00189 BC00189 V=166.7  +MOVJ EC00189
SMOVL C00190 BC00190 V=166.7  +MOVJ EC00190
SREFP 3 C00191 BC00191  +REFP EC00191
CALL JOB:SEARCH-R1-S13D
SET P022 P006
SFTON3D P022
SMOVL C00192 BC00192 V=166.7  +MOVJ EC00192
SMOVL C00193 BC00193 V=166.7  +MOVJ EC00193
SMOVL C00194 BC00194 V=166.7  +MOVJ EC00194
MOVL C00195 BC00195 V=800.0  +MOVJ EC00195 VJ=100.00
MOVL C00196 BC00196 V=1000.0  +MOVJ EC00196 VJ=100.00
'EndPath S4742
MOVJ C00197 BC00197 VJ=100.00  +MOVJ EC00197 VJ=100.00
MOVJ C00198 BC00198 VJ=100.00  +MOVJ EC00198 VJ=100.00
'Path S4741
SFTOF3D
MOVJ C00199 BC00199 VJ=100.00  +MOVJ EC00199 VJ=100.00
MOVL C00200 BC00200 V=800.0  +MOVJ EC00200 VJ=100.00
SMOVL C00201 BC00201 V=166.7  +MOVJ EC00201
SREFP 3 C00202 BC00202  +REFP EC00202
CALL JOB:SEARCH-R1-S13D
SET P021 P006
SFTON3D P021
SMOVL C00203 BC00203 V=166.7  +MOVJ EC00203
SMOVL C00204 BC00204 V=166.7  +MOVJ EC00204
SREFP 3 C00205 BC00205  +REFP EC00205
CALL JOB:SEARCH-R1-S13D
SET P021 P006
SFTON3D P021
SMOVL C00206 BC00206 V=166.7  +MOVJ EC00206
SMOVL C00207 BC00207 V=166.7  +MOVJ EC00207
SMOVL C00208 BC00208 V=166.7  +MOVJ EC00208
SREFP 3 C00209 BC00209  +REFP EC00209
CALL JOB:SEARCH-R1-S13D
SET P021 P006
SFTON3D P021
SMOVL C00210 BC00210 V=166.7  +MOVJ EC00210
SMOVL C00211 BC00211 V=166.7  +MOVJ EC00211
SMOVL C00212 BC00212 V=166.7  +MOVJ EC00212
MOVL C00213 BC00213 V=800.0  +MOVJ EC00213 VJ=100.00
MOVL C00214 BC00214 V=1000.0  +MOVJ EC00214 VJ=100.00
'EndPath S4741
'Path W4746
SFTOF3D
SFTON3D P021
MOVJ C00215 BC00215 VJ=100.00  +MOVJ EC00215 VJ=100.00
SMOVL C00216 BC00216 V=800.0  +MOVJ EC00216
SMOVL C00217 BC00217 V=150.0 PL=0  +MOVJ EC00217
ARCON
SMOVL C00218 BC00218 V=11.7  +MOVJ EC00218
SMOVL C00219 BC00219 V=11.7  +MOVJ EC00219
SMOVL C00220 BC00220 V=12.5  +MOVJ EC00220
SMOVL C00221 BC00221 V=12.5  +MOVJ EC00221
SMOVL C00222 BC00222 V=12.5  +MOVJ EC00222
ARCOF
SMOVL C00223 BC00223 V=800.0  +MOVJ EC00223
SMOVL C00224 BC00224 V=1000.0  +MOVJ EC00224
SFTOF3D
'EndPath W4746
MOVJ C00225 BC00225 VJ=100.00  +MOVJ EC00225 VJ=100.00
MOVJ C00226 BC00226 VJ=100.00  +MOVJ EC00226 VJ=100.00
'Path W4747
SFTOF3D
SFTON3D P022
MOVJ C00227 BC00227 VJ=100.00  +MOVJ EC00227 VJ=100.00
SMOVL C00228 BC00228 V=800.0  +MOVJ EC00228
SMOVL C00229 BC00229 V=150.0 PL=0  +MOVJ EC00229
ARCON
SMOVL C00230 BC00230 V=10.0  +MOVJ EC00230
SMOVL C00231 BC00231 V=10.0  +MOVJ EC00231
SMOVL C00232 BC00232 V=10.0  +MOVJ EC00232
ARCOF
SMOVL C00233 BC00233 V=800.0  +MOVJ EC00233
SMOVL C00234 BC00234 V=1000.0  +MOVJ EC00234
SFTOF3D
'EndPath W4747
MOVJ C00235 BC00235 VJ=100.00  +MOVJ EC00235 VJ=100.00
MOVJ C00236 BC00236 VJ=100.00  +MOVJ EC00236 VJ=100.00
'Path W4748
SFTOF3D
SFTON3D P023
MOVJ C00237 BC00237 VJ=100.00  +MOVJ EC00237 VJ=100.00
SMOVL C00238 BC00238 V=800.0  +MOVJ EC00238
SMOVL C00239 BC00239 V=150.0 PL=0  +MOVJ EC00239
ARCON
SMOVL C00240 BC00240 V=10.0  +MOVJ EC00240
SMOVL C00241 BC00241 V=10.0  +MOVJ EC00241
SMOVL C00242 BC00242 V=10.8  +MOVJ EC00242
SFTON3D P024
SMOVL C00243 BC00243 V=10.8  +MOVJ EC00243
SMOVL C00244 BC00244 V=10.8  +MOVJ EC00244
SMOVL C00245 BC00245 V=10.8  +MOVJ EC00245
SMOVL C00246 BC00246 V=10.8  +MOVJ EC00246
SMOVL C00247 BC00247 V=10.0  +MOVJ EC00247
SMOVL C00248 BC00248 V=10.0  +MOVJ EC00248
ARCOF
SMOVL C00249 BC00249 V=800.0  +MOVJ EC00249
SMOVL C00250 BC00250 V=1000.0  +MOVJ EC00250
SFTOF3D
'EndPath W4748
MOVJ C00251 BC00251 VJ=100.00  +MOVJ EC00251 VJ=100.00
MOVJ C00252 BC00252 VJ=100.00  +MOVJ EC00252 VJ=100.00
'Path W4749
SFTOF3D
SFTON3D P025
MOVJ C00253 BC00253 VJ=100.00  +MOVJ EC00253 VJ=100.00
SMOVL C00254 BC00254 V=800.0  +MOVJ EC00254
SMOVL C00255 BC00255 V=150.0 PL=0  +MOVJ EC00255
ARCON
SMOVL C00256 BC00256 V=9.2  +MOVJ EC00256
SMOVL C00257 BC00257 V=9.2  +MOVJ EC00257
ARCOF
SMOVL C00258 BC00258 V=800.0  +MOVJ EC00258
SMOVL C00259 BC00259 V=1000.0  +MOVJ EC00259
SFTOF3D
'EndPath W4749
MOVJ C00260 BC00260 VJ=100.00  +MOVJ EC00260 VJ=100.00
MOVJ C00261 BC00261 VJ=100.00  +MOVJ EC00261 VJ=100.00
MOVJ C00262 BC00262 VJ=100.00  +MOVJ EC00262 VJ=100.00
CALL JOB:CLEAN-R1_KM_NEW
MOVJ C00263 BC00263 VJ=50.00  +MOVJ EC00263 VJ=50.00
'
'
'
MOVJ C00264 BC00264 VJ=100.00  +MOVJ EC00264 VJ=100.00
'Path S4750
SFTOF3D
MOVJ C00265 BC00265 VJ=100.00  +MOVJ EC00265 VJ=100.00
MOVL C00266 BC00266 V=800.0  +MOVJ EC00266 VJ=100.00
SMOVL C00267 BC00267 V=166.7  +MOVJ EC00267
SREFP 3 C00268 BC00268  +REFP EC00268
CALL JOB:SEARCH-R1-S13D
SET P035 P006
SFTON3D P035
SMOVL C00269 BC00269 V=166.7  +MOVJ EC00269
SMOVL C00270 BC00270 V=166.7  +MOVJ EC00270
SREFP 3 C00271 BC00271  +REFP EC00271
CALL JOB:SEARCH-R1-S13D
SET P035 P006
SFTON3D P035
SMOVL C00272 BC00272 V=166.7  +MOVJ EC00272
SMOVL C00273 BC00273 V=166.7  +MOVJ EC00273
SREFP 3 C00274 BC00274  +REFP EC00274
CALL JOB:SEARCH-R1-S13D
SET P035 P006
SFTON3D P035
SMOVL C00275 BC00275 V=166.7  +MOVJ EC00275
MOVL C00276 BC00276 V=800.0  +MOVJ EC00276 VJ=100.00
MOVL C00277 BC00277 V=1000.0  +MOVJ EC00277 VJ=100.00
'EndPath S4750
'Path S4751
SFTOF3D
MOVJ C00278 BC00278 VJ=100.00  +MOVJ EC00278 VJ=100.00
MOVL C00279 BC00279 V=800.0  +MOVJ EC00279 VJ=100.00
SMOVL C00280 BC00280 V=166.7  +MOVJ EC00280
SREFP 3 C00281 BC00281  +REFP EC00281
CALL JOB:SEARCH-R1-S13D
SET P034 P006
SFTON3D P034
SMOVL C00282 BC00282 V=166.7  +MOVJ EC00282
SMOVL C00283 BC00283 V=166.7  +MOVJ EC00283
SREFP 3 C00284 BC00284  +REFP EC00284
CALL JOB:SEARCH-R1-S13D
SET P034 P006
SFTON3D P034
SMOVL C00285 BC00285 V=166.7  +MOVJ EC00285
MOVL C00286 BC00286 V=800.0  +MOVJ EC00286 VJ=100.00
MOVL C00287 BC00287 V=1000.0  +MOVJ EC00287 VJ=100.00
'EndPath S4751
'Path S4752
SFTOF3D
MOVJ C00288 BC00288 VJ=100.00  +MOVJ EC00288 VJ=100.00
MOVL C00289 BC00289 V=800.0  +MOVJ EC00289 VJ=100.00
SMOVL C00290 BC00290 V=166.7  +MOVJ EC00290
SREFP 3 C00291 BC00291  +REFP EC00291
CALL JOB:SEARCH-R1-S13D
SET P033 P006
SFTON3D P033
SMOVL C00292 BC00292 V=166.7  +MOVJ EC00292
SMOVL C00293 BC00293 V=166.7  +MOVJ EC00293
SREFP 3 C00294 BC00294  +REFP EC00294
CALL JOB:SEARCH-R1-S13D
SET P033 P006
SFTON3D P033
SMOVL C00295 BC00295 V=166.7  +MOVJ EC00295
MOVL C00296 BC00296 V=800.0  +MOVJ EC00296 VJ=100.00
MOVL C00297 BC00297 V=1000.0  +MOVJ EC00297 VJ=100.00
'EndPath S4752
'Path S4753
SFTOF3D
MOVJ C00298 BC00298 VJ=100.00  +MOVJ EC00298 VJ=100.00
MOVL C00299 BC00299 V=800.0  +MOVJ EC00299 VJ=100.00
SMOVL C00300 BC00300 V=166.7  +MOVJ EC00300
SREFP 3 C00301 BC00301  +REFP EC00301
CALL JOB:SEARCH-R1-S13D
SET P032 P006
SFTON3D P032
SMOVL C00302 BC00302 V=166.7  +MOVJ EC00302
SMOVL C00303 BC00303 V=166.7  +MOVJ EC00303
SREFP 3 C00304 BC00304  +REFP EC00304
CALL JOB:SEARCH-R1-S13D
SET P032 P006
SFTON3D P032
SMOVL C00305 BC00305 V=166.7  +MOVJ EC00305
MOVL C00306 BC00306 V=800.0  +MOVJ EC00306 VJ=100.00
MOVL C00307 BC00307 V=1000.0  +MOVJ EC00307 VJ=100.00
'EndPath S4753
'Path S4754
SFTOF3D
MOVJ C00308 BC00308 VJ=100.00  +MOVJ EC00308 VJ=100.00
MOVL C00309 BC00309 V=800.0  +MOVJ EC00309 VJ=100.00
SMOVL C00310 BC00310 V=166.7  +MOVJ EC00310
SREFP 3 C00311 BC00311  +REFP EC00311
CALL JOB:SEARCH-R1-S13D
SET P032 P006
SFTON3D P032
SMOVL C00312 BC00312 V=166.7  +MOVJ EC00312
SMOVL C00313 BC00313 V=166.7  +MOVJ EC00313
SREFP 3 C00314 BC00314  +REFP EC00314
CALL JOB:SEARCH-R1-S13D
SET P032 P006
SFTON3D P032
SMOVL C00315 BC00315 V=166.7  +MOVJ EC00315
MOVL C00316 BC00316 V=800.0  +MOVJ EC00316 VJ=100.00
MOVL C00317 BC00317 V=1000.0  +MOVJ EC00317 VJ=100.00
'EndPath S4754
'Path S4756
SFTOF3D
MOVJ C00318 BC00318 VJ=100.00  +MOVJ EC00318 VJ=100.00
MOVL C00319 BC00319 V=800.0  +MOVJ EC00319 VJ=100.00
SMOVL C00320 BC00320 V=166.7  +MOVJ EC00320
SREFP 3 C00321 BC00321  +REFP EC00321
CALL JOB:SEARCH-R1-S13D
SET P031 P006
SFTON3D P031
SMOVL C00322 BC00322 V=166.7  +MOVJ EC00322
SMOVL C00323 BC00323 V=166.7  +MOVJ EC00323
SREFP 3 C00324 BC00324  +REFP EC00324
CALL JOB:SEARCH-R1-S13D
SET P031 P006
SFTON3D P031
SMOVL C00325 BC00325 V=166.7  +MOVJ EC00325
SMOVL C00326 BC00326 V=166.7  +MOVJ EC00326
SREFP 3 C00327 BC00327  +REFP EC00327
CALL JOB:SEARCH-R1-S13D
SET P031 P006
SFTON3D P031
SMOVL C00328 BC00328 V=166.7  +MOVJ EC00328
MOVL C00329 BC00329 V=800.0  +MOVJ EC00329 VJ=100.00
MOVL C00330 BC00330 V=1000.0  +MOVJ EC00330 VJ=100.00
'EndPath S4756
'Path W4751
SFTOF3D
SFTON3D P032
MOVJ C00331 BC00331 VJ=100.00  +MOVJ EC00331 VJ=100.00
SMOVL C00332 BC00332 V=800.0  +MOVJ EC00332
SMOVL C00333 BC00333 V=150.0 PL=0  +MOVJ EC00333
MACRO1 MJ#(0) ARGF21
ARCON
SFTON3D P031
SMOVL C00334 BC00334 V=7.5  +MOVJ EC00334
SMOVL C00335 BC00335 V=7.5  +MOVJ EC00335
ARCOF
SMOVL C00336 BC00336 V=800.0  +MOVJ EC00336
SMOVL C00337 BC00337 V=1000.0  +MOVJ EC00337
SFTOF3D
'EndPath W4751
'Path W4755
SFTOF3D
SFTON3D P034
MOVJ C00338 BC00338 VJ=100.00  +MOVJ EC00338 VJ=100.00
SMOVL C00339 BC00339 V=800.0  +MOVJ EC00339
SMOVL C00340 BC00340 V=150.0 PL=0  +MOVJ EC00340
ARCON
SFTON3D P035
SMOVL C00341 BC00341 V=7.5  +MOVJ EC00341
SMOVL C00342 BC00342 V=7.5  +MOVJ EC00342
ARCOF
SMOVL C00343 BC00343 V=800.0  +MOVJ EC00343
SMOVL C00344 BC00344 V=1000.0  +MOVJ EC00344
SFTOF3D
'EndPath W4755
'Path W4752
SFTOF3D
SFTON3D P032
MOVJ C00345 BC00345 VJ=100.00  +MOVJ EC00345 VJ=100.00
SMOVL C00346 BC00346 V=800.0  +MOVJ EC00346
SMOVL C00347 BC00347 V=150.0 PL=0  +MOVJ EC00347
ARCON
SFTON3D P033
SMOVL C00348 BC00348 V=7.5  +MOVJ EC00348
ARCOF
SMOVL C00349 BC00349 V=800.0  +MOVJ EC00349
SMOVL C00350 BC00350 V=1000.0  +MOVJ EC00350
SFTOF3D
'EndPath W4752
'Path W4754
SFTOF3D
SFTON3D P034
MOVJ C00351 BC00351 VJ=100.00  +MOVJ EC00351 VJ=100.00
SMOVL C00352 BC00352 V=800.0  +MOVJ EC00352
SMOVL C00353 BC00353 V=150.0 PL=0  +MOVJ EC00353
ARCON
SFTON3D P033
SMOVL C00354 BC00354 V=8.3  +MOVJ EC00354
SMOVL C00355 BC00355 V=8.3  +MOVJ EC00355
ARCOF
SMOVL C00356 BC00356 V=800.0  +MOVJ EC00356
SMOVL C00357 BC00357 V=1000.0  +MOVJ EC00357
SFTOF3D
SMOVL C00358 BC00358 V=1000.0  +MOVJ EC00358
SMOVL C00359 BC00359 V=1000.0  +MOVJ EC00359
SMOVL C00360 BC00360 V=1000.0  +MOVJ EC00360
SMOVL C00361 BC00361 V=1000.0  +MOVJ EC00361
SMOVL C00362 BC00362 V=250.0  +MOVJ EC00362
ARCON
SMOVL C00363 BC00363 V=8.3  +MOVJ EC00363
SFTON3D P031
SMOVL C00364 BC00364 V=8.3  +MOVJ EC00364
ARCOF
SMOVL C00365 BC00365 V=250.0  +MOVJ EC00365
SMOVL C00366 BC00366 V=250.0  +MOVJ EC00366
SMOVL C00367 BC00367 V=250.0  +MOVJ EC00367
SMOVL C00368 BC00368 V=250.0  +MOVJ EC00368
ARCON
SMOVL C00369 BC00369 V=8.3  +MOVJ EC00369
SMOVL C00370 BC00370 V=8.3  +MOVJ EC00370
ARCOF
SMOVL C00371 BC00371 V=250.0  +MOVJ EC00371
SFTOF3D
'EndPath W4754
MOVJ C00372 BC00372 VJ=100.00  +MOVJ EC00372 VJ=100.00
MOVJ C00373 BC00373 VJ=100.00  +MOVJ EC00373 VJ=100.00
MOVJ C00374 BC00374 VJ=100.00  +MOVJ EC00374 VJ=100.00
MOVJ C00375 BC00375 VJ=15.00  +MOVJ EC00375 VJ=100.00
SFTON3D P035
SMOVL C00376 BC00376 V=166.7  +MOVJ EC00376
ARCON
SMOVL C00377 BC00377 V=8.3  +MOVJ EC00377
SMOVL C00378 BC00378 V=8.3  +MOVJ EC00378
SMOVL C00379 BC00379 V=8.3  +MOVJ EC00379
ARCOF
MOVJ C00380 BC00380 VJ=100.00  +MOVJ EC00380 VJ=100.00
MOVJ C00381 BC00381 VJ=100.00  +MOVJ EC00381 VJ=100.00
SMOVL C00382 BC00382 V=166.7  +MOVJ EC00382
ARCON
SMOVL C00383 BC00383 V=7.5  +MOVJ EC00383
SMOVL C00384 BC00384 V=7.5  +MOVJ EC00384
ARCOF
SMOVL C00385 BC00385 V=166.7  +MOVJ EC00385
SMOVL C00386 BC00386 V=166.7  +MOVJ EC00386
SFTOF3D
MOVJ C00387 BC00387 VJ=100.00  +MOVJ EC00387 VJ=100.00
MOVJ C00388 BC00388 VJ=100.00  +MOVJ EC00388 VJ=100.00
END
